PROGRAM PRG_1_PlcTask
VAR

bDebug : Bool := FALSE;
bMotionTest : Bool := FALSE;
fbLogHandler: FB_LogHandler;
	
END_VAR

(*Ethercat Diagnostics*)
DIAGNOSTICS();
// Vacuum and differential pumping
PRG_GATT();
// Injector
PRG_INJ();

if (NOT bDebug)Then
	// Motorised valve
	PRG_VGP();
END_IF
if (NOT bMotionTest)Then
	// Functionblock for PTP motion between different appertures
	PRG_Motion();
ELSE
	PRG_Motors_Test();
END_IF

PRG_ILK();

//Logger
fbLogHandler();

END_PROGRAM

(* stored: Version 1.1.0.1, ProductVersion 3.1.4022.18
   POU PRG_1_PlcTask: Id {974f2793-1abb-41d3-ab47-a860d1c380f6}, SpecialFunc None *)
